VAR_GLOBAL
	bRemote:BOOL:=TRUE;
END_VAR

(* stored: Version 1.1.0.1, ProductVersion 3.1.4022.18
   GVL GVL_Remote: Id {10367ee5-1a8c-4e85-b1f2-1ccf36d7dd66} *)
